// TIA Portal V20 export
VAR_GLOBAL   // PLC tag table "Constantes de Maquinas"
END_VAR
VAR_GLOBAL CONSTANT   // user constants
   CTE_TipoMaquinaVTDC : UInt := 74;
   CTE_TipoMaquinaELEV : UInt := 71;
   CTE_TipoMaquina : UInt := 70;
   CTE_TipoMaquinaREMO : UInt := 72;
   CTE_TipoMaquinaAPIL : UInt := 73;
   CTE_TipoMaquinaENFA : UInt := 75;
   CTE_TipoMaquinaETIQ : UInt := 76;
   CTE_TipoMaquinaFLEJ : UInt := 77;
   CTE_OperacionSTAT : UInt := 5000;
   CTE_OperacionPOSI : UInt := 5001;
   TIPO_MAQ_PANTALLA_APIL_DESAPIL_PALETAS : USInt := 100;
   TIPO_MAQ_PANTALLA_REMONTADOR : USInt := 101;
   TIPO_MAQ_PANTALLA_ELEVADOR : USInt := 102;
   TIPO_MAQ_PANTALLA_CTS : USInt := 103;
   TIPO_MAQ_PANTALLA_APIL_BANDEJAS : USInt := 104;
   TIPO_MAQ_PANTALLA_DESAPIL_BANDEJAS : USInt := 105;
   TIPO_MAQ_PANTALLA_APIL_ERAMAN : USInt := 106;
   TIPO_MAQ_PANTALLA_DESAPIL_ERAMAN : USInt := 107;
   "TIPO_INTERLOCK_CS/FS" : USInt := 150;
   TIPO_INTERLOCK_FSS : USInt := 151;
   TIPO_INTERLOCK_STV : USInt := 152;
   TIPO_INTERLOCK_ZETES : USInt := 153;
   TIPO_INTERLOCK_AMR : USInt := 154;
   TIPO_INTERLOCK_PUERTA_RF : USInt := 155;
   TIPO_INTERLOCK_PUERTA_RAPIDA : USInt := 156;
   TIPO_INTERLOCK_FLEJADORA : USInt := 157;
   TIPO_INTERLOCK_ENFARDADORA : USInt := 158;
   TIPO_INTERLOCK_HAI : USInt := 159;
   TIPO_MESA_ESTANDAR : USInt := 50;
   TIPO_MESA_FSS : USInt := 54;
   TIPO_MESA_MAQUETAS : USInt := 99;
END_VAR
